RESOURCE_TYPE EMB_RES2 (* An Embedded Resource Type with a FBD installed *)
  (* Standard: 61499-1; Function: Device Management; Description: A simple embedded resource *)
  (* Version 0.0, 2001-01-04, JHC, Rockwell Automation *)
  (* Compiler header: import fb.rt.math.*; *)
  (* Compiler Java IBM VisualAge 3.0 *)
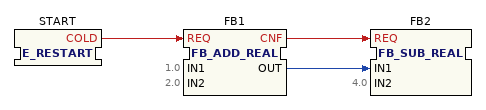
  FBS
    START : E_RESTART;
    FB1 : FB_ADD_REAL(IN1 := 1.0, IN2 := 2.0);
    FB2 : FB_SUB_REAL(IN2 := 4.0);
  END_FBS
  EVENT_CONNECTIONS
    START.COLD TO FB1.REQ;
    FB1.CNF TO FB2.REQ;
  END_CONNECTIONS
  DATA_CONNECTIONS
    FB1.OUT TO FB2.IN1;
  END_CONNECTIONS
END_RESOURCE_TYPE
